Universal Robots URScript: andrea7.script

def andrea7():
  set_safety_mode_transition_hardness(1)
  set_tcp(p[-0.0475,0.08227,0.045,0.0,0.0,0.0])
  set_payload(2.6)
  set_tool_voltage(0)
  set_standard_analog_input_domain(0, 1)
  set_standard_analog_input_domain(1, 1)
  set_tool_analog_input_domain(0, 1)
  set_tool_analog_input_domain(1, 1)
  set_analog_outputdomain(0, 0)
  set_analog_outputdomain(1, 0)
  set_input_actions_to_default()
  set_gravity([8.503688472232543E-16, 6.943788591251896, 6.943788591251898])
  step_count_136e9950_01e8_4336_b553_866481468409 = 0.0
  thread Step_Counter_Thread_6807c733_f62a_40d3_b02d_d4e106b82d18():
    while (True):
      step_count_136e9950_01e8_4336_b553_866481468409 = step_count_136e9950_01e8_4336_b553_866481468409 + 1.0
      sync()
    end
  end
  run Step_Counter_Thread_6807c733_f62a_40d3_b02d_d4e106b82d18()
  global Piano_Carrello=p[0.15738038194676504,0.34804679499613556,-0.10180660081110104,-0.604770547029434,0.6135130099633843,1.4699264996051509]
  global Piano_Inclinato=p[0.24163290852284977,0.484348843812812,-0.08183038406600258,-0.13450397856501406,0.1337107555826035,1.5511152546959441]
  global piano_moduli=p[0.13993944179688836,0.3246186948043025,-0.2543011639693953,-0.6047704836459776,0.6135130132010319,1.4699264397811034]
  global XY=[0,0]
  global ant=3
  global col=4
  global ghr=2
  global nCycle=0
  global nfc=1
  global pallStocks=[16,16,16,40,16,16,16,40,16,16,16,40,16,40,0,0]
  global pick=[0,0]
  while (True):
    $ 2 "Robot Program"
    $ 3 "Script: relPose.script_bak"
    def relPose(FeaturePose,vect):

        # FeaturePose is the pose for the feature
        # vect = p[0.1, 0, 0, 0, 0, 0] makes us move 10cm in the X direction of the feature
        # credits: https://forum.universal-robots.com/t/move-tcp-relative-to-feature/15492

       PoseRelativeToFeature = pose_trans(pose_inv(FeaturePose), get_actual_tcp_pose())
       MoveTCPRelativeToFeature = pose_add(PoseRelativeToFeature, vect)
       return pose_trans(FeaturePose, MoveTCPRelativeToFeature)

    end
    $ 4 "Script: calcItemPosition.script"
    def calcItemPosition(pick, item, pallDefs, grid, featOrigin):

        # calcola la posizione assoluta del pezzo scelto da pickPalletItem

        # nPosX è il numero di colonne
        # nPosY è il numero di righe
        # distX è la distanza tra colonne
        # distY è la distanza tra righe
        # [posX1, posY1] è la posizione del primo pezzo rispetto all'origine del pallet

        nPallet = pick[0] + 1 # numero del pallet (gli id partono da 0)
        nItem = pick[1] + 1 # numero del pezzo

        nPosXgrid = grid[0] # numero di posizioni della giglia in X
        distXgrid = grid[2] # distanza tra gli slot della griglia in X
        distYgrid = grid[3] # distanza tra gli slot della griglia in Y

        pallPosX = nPallet%nPosXgrid
        if(pallPosX==0): pallPosX = nPosXgrid end
        pallPosY = ceil(nPallet/nPosXgrid)

        pallPosX1 = grid[4]
        pallPosY1 = grid[5]


        nPosX = pallDefs[item,0]
        nPosY = pallDefs[item,1]
        distX = pallDefs[item,2]
        distY = pallDefs[item,3]
        posX1 = pallDefs[item,4]
        posY1 = pallDefs[item,5]

        posX = nItem%nPosX
        if(posX==0): posX = nPosX end
        posY = ceil(nItem/nPosX)

        # [X,Y] è la posizione del pezzo rispetto all'origine della griglia

        X=distX*(posX - 1) + posX1 + distXgrid*(pallPosX - 1) + pallPosX1
        Y=distY*(posY - 1) + posY1 + distYgrid*(pallPosY - 1) + pallPosY1
        xy=[X,Y]

        return xy

     end
    $ 5 "Script: pickPalletItem.script_bak"
    def pickPalletItem(type, pallDefs, pallTypes, pallStocks):

      # seleziona un pezzo sulla griglia, noti il tipo di pezzo e lo stato della griglia

      # lo script funziona finché le variabili del robot non vengono resettate. Tuttavia, anche
      # in caso di riavvio, è possibile scrivere manualmente le info sulla griglia e lo stock
      # all'inizio del programma, così da 'insegnare' al robot dove farlo
      # riprendere

      iPallet = 0 # inizializzo l'id del pallet

      while iPallet < length(pallStocks):

        if pallTypes[iPallet] == type and pallStocks[iPallet] > 0 :

          nItems = pallStocks[iPallet] # numero di pezzi nello stock del pallet iesimo

          nPosX = pallDefs[type,0] # numero di posizioni lungo x, come definito per il pallet di tipo "type"
          nPosY = pallDefs[type,1] # numero di posizioni lungo y, come definito per il pallet di tipo "type"

          stockMax = nPosX*nPosY
          iItem = stockMax - nItems # id del pezzo

          pick = [iPallet,iItem]

          # pick = [id del pallet, id del pezzo]

          return pick
     end
    iPallet = iPallet + 1
    end
    end
    $ 6 "Script: stockUpdate.script_bak"
    def stockUpdate(pick,stock):

        # simple function that ingests the output of pickItem and returns the
        # modified stock array. just so to avoid using global variables and
        # multi-dimensional arrays

        i = pick[0]
        stock[i] = stock[i] - 1
        return stock


    end
    $ 7 "Script: ini_grid.script"
    def ini_grid():

        # grid = [nPallPosX, nPallPosY, distPallX, distPallY, pallPosX1, pallPosY1, pallPosZ1]
        # la struttura e' del tutto analoga in logica con quella espressa in defs
        grid = [4, 4, 90, 90, 10, 20, 6]
        return grid
    end
    $ 8 "Script: ini_defs.script"
    def ini_defs():

        # definition = [nPosX,nPosY,distX,distY,posX1,posY1,posZ1]

        # nPosX è il numero di colonne
        # nPosY è il numero di righe
        # distX è la distanza tra colonne
        # distY è la distanza tra righe
        # [posX1, posY1] è la posizione del primo pezzo rispetto all'origine del pallet
        # posZ1 e' la posizione che deve raggiungere il TCP lungo asse Z, che sarebbe asse verticale

        defs = [
            [0, 0, 0, 0, 0, 0, 0], # slot vuoto
            [4, 10, 18, 8, 17.5, 5.7, 11.1], # pallet nfc
            [4, 4, 21, 21, 12.5, 12.5, 49], # pallet ghiere
            [1, 1, 0, 0, 132.06, 44, 16.05], # stazione antenna
            [1, 2, 0, 40, 20.256, 24, 27.85] # stazione incollaggio
        ]
        return defs
    end
    $ 9 "Script: ini_types.script_bak"
    def ini_types():

        visualTypes = [

            [0,0,0,0],
            [ghr,0,0,0],
            [0,0,nfc,0],
            [0,0,0,0]

        ]

    # purtroppo fare questa array vuota di dimensione (righe)x(colonne) per aggirare le limitazioni di UR
    # bisogna ricordarsi di cambiare questa dichiarazione di types se si cambia dimensione griglia

         types = [0,0,0,0,0,0,0,0,0,0,0,0,0,0,0,0]

        iii = 0
        s = size(visualTypes)
        i = 0
        while i < s[0]:

            ii=0
            while ii < s[1]:

                types[iii] = visualTypes[s[0]-1-i,ii]
                ii = ii + 1
                iii = iii + 1
            end
        i = i + 1
        end
        return types
    end
    $ 10 "Script: ini_stocks.script_bak_bak"
    def ini_stocks(defs, types):

        global f = -1 # usa questo carattere per inizializzare automaticamente pallet pieni

        visualStocks = [

            [f, f, f, f],
            [f, f, f, f],
            [f, f, f, f],
            [f ,f, f, f]

        ]

    # purtroppo fare questa array vuota di dimensione (righe)x(colonne) per aggirare le limitazioni di UR
    # bisogna ricordarsi di cambiare questa dichiarazione di types se si cambia dimensione griglia

         stocks = [0,0,0,0,0,0,0,0,0,0,0,0,0,0,0,0]

        iii = 0
        s = size(visualStocks)
        i = 0
        while i < s[0]:

            ii=0
            while ii < s[1]:
                if visualStocks[s[0]-1-i,ii] == f:
                    nPosX = defs[types[iii], 0]
                    nPosY = defs[types[iii], 1]
                    stocks[iii] = nPosX*nPosY
                else:

                    stocks[iii] = visualStocks[s[0]-1-i,ii]
                end
                ii = ii + 1
                iii = iii + 1
            end
        i = i + 1
        end
        return stocks
    end
    $ 11 "If nCycle≟0"
    if (nCycle == 0):
      $ 12 "pallTypes≔ini_types()"
      global pallTypes=ini_types()
      $ 13 "grid≔ini_grid()"
      global grid=ini_grid()
      $ 14 "pallDefs≔ini_defs()"
      global pallDefs=ini_defs()
      $ 15 "pallStocks≔ini_stocks(pallDefs,pallTypes)"
      global pallStocks=ini_stocks(pallDefs,pallTypes)
      $ 17 "nCycle≔1"
      global nCycle=1
      $ 18 "ghr≔ghr"
      global ghr=ghr
      $ 19 "nfc≔nfc"
      global nfc=nfc
      $ 20 "ant≔ant"
      global ant=ant
      $ 21 "col≔col"
      global col=col
    end
    $ 22 "MoveJ"
    $ 24 "azzeramento" "breakAfter"
    set_tcp(p[-0.0475,0.08227,0.045,0.0,0.0,0.0])
    movej(get_inverse_kin(p[.035262995133, .412914797501, -.175544399089, -2.288575391083, -.604632993317, -.263002031178], qnear=[-1.947583023701803, -0.8369515577899378, 1.9894261360168457, -0.3385861555682581, 1.3188148736953735, 2.3547770977020264]), a=1.3962634015954636, v=1.0471975511965976)
    $ 25 "item≔1"
    global item=1
    $ 26 "pick≔pickPalletItem(item,pallDefs,pallTypes,pallStocks)"
    global pick=pickPalletItem(item,pallDefs,pallTypes,pallStocks)
    $ 27 "Popup"
    popup(str_cat("",pick), "Message", False, False, blocking=True)
    $ 28 "XY≔calcItemPosition(pick, item,pallDefs, grid)"
    global XY=calcItemPosition(pick, item,pallDefs, grid)
    $ 29 "MoveJ"
    $ 30 "Popup"
    popup(str_cat("",XY), "Message", False, False, blocking=True)
    $ 32 "p_pall≔relPose(piano_moduli,p[XY[0]/1000,XY[1]/1000,0.0,0.0,0.0,0.0])"
    global p_pall=relPose(piano_moduli,p[XY[0]/1000,XY[1]/1000,0.0,0.0,0.0,0.0])
    $ 33 "p_pall" "breakAfter"
    set_tcp(p[-0.0475,0.08227,0.045,0.0,0.0,0.0])
    movej(p_pall, a=1.3962634015954636, v=1.0471975511965976)
    $ 37 "MoveL"
    $ 39 "p_pall≔relPose(Piano_Carrello_const,p[0.0,0.0,-0.09,0.0,0.0,0.0])"
    global p_pall=relPose(p[0.15738038194676504,0.34804679499613556,-0.10180660081110104,-0.604770547029434,0.6135130099633843,1.4699264996051509],p[0.0,0.0,-0.09,0.0,0.0,0.0])
    $ 40 "p_pall" "breakAfter"
    set_tcp(p[-0.0475,0.08227,0.045,0.0,0.0,0.0])
    movel(pose_trans(p[0.0,0.0,0.0,0.0,0.0,0.0], p_pall), a=1.2, v=0.25)
    $ 41 "p_pall≔relPose(Piano_Carrello_const,p[0.0,0.0,+0.09,0.0,0.0,0.0])"
    global p_pall=relPose(p[0.15738038194676504,0.34804679499613556,-0.10180660081110104,-0.604770547029434,0.6135130099633843,1.4699264996051509],p[0.0,0.0,+0.09,0.0,0.0,0.0])
    $ 42 "p_pall" "breakAfter"
    set_tcp(p[-0.0475,0.08227,0.045,0.0,0.0,0.0])
    movel(pose_trans(p[0.0,0.0,0.0,0.0,0.0,0.0], p_pall), a=1.2, v=0.25)
    $ 43 "pallStocks≔stockUpdate(pick,pallStocks)"
    global pallStocks=stockUpdate(pick,pallStocks)
    $ 44 "Popup"
    popup(str_cat("",pallStocks), "Message", False, False, blocking=True)
  end
end
